{attribute 'linkalways'} 
{attribute 'no_explicit_call' := 'This FB is a CLASS and must be accessed using methods or properties'}
{attribute 'enable_dynamic_creation'}
FUNCTION_BLOCK _WORD EXTENDS DatatypeBase
VAR
	localData : WORD;
	activeData : REFERENCE TO WORD REF= localData;
END_VAR

PROPERTY PUBLIC Address : PVOID
GET
Address := ADR(activeData);
END_GET
END_PROPERTY

METHOD PUBLIC ClearReference
VAR_INPUT
END_VAR
activeData REF= localData;
END_METHOD

METHOD PUBLIC Clone : I_Datatype
VAR
    pClone : POINTER TO _WORD;
END_VAR
pClone := __NEW(_WORD(InitialValue := Value));
Clone := pClone^;
END_METHOD

METHOD FB_init : BOOL
VAR_INPUT
	bInitRetains : BOOL; // if TRUE, the retain variables are initialized (warm start / cold start)
	bInCopyCode : BOOL;  // if TRUE, the instance afterwards gets moved WORDo the copy code (online change)
	InitialValue : WORD;
END_VAR
localData := InitialValue;
END_METHOD

PROPERTY PUBLIC IecType : T_MAXSTRING
GET
IecType := 'WORD';
END_GET
END_PROPERTY

METHOD PUBLIC MakeReferenceTo
VAR_INPUT
	ReferenceTarget : REFERENCE TO WORD;
END_VAR
activeData REF= ReferenceTarget;
END_METHOD

METHOD PUBLIC SerializeWith
VAR_INPUT
	Serializer : I_Serializer;
END_VAR
Serializer.AddWord(activeData);
END_METHOD

PROPERTY PUBLIC Size : UDINT
GET
Size := SIZEOF(activeData);
END_GET
END_PROPERTY

METHOD TryDeserializeFrom : BOOL
VAR_INPUT
	Deserializer : I_Deserializer;
	Feedback : I_DeserializerFeedback;
END_VAR
TryDeserializeFrom := Deserializer.TryGetWord(activeData, Feedback);
END_METHOD

METHOD TryMakeReferenceTo : BOOL
VAR_INPUT
	Target : I_Datatype;
END_VAR
VAR
	pTargetData : POINTER TO WORD;
END_VAR
IF NOT (Target.IecType = IecType) THEN
	RETURN;
END_IF

pTargetData := Target.Address;
activeData REF= pTargetData^;
TryMakeReferenceTo := TRUE;
END_METHOD

PROPERTY PUBLIC Value : WORD
GET
Value := activeData;
END_GET
SET
activeData := Value;
END_SET
END_PROPERTY

END_FUNCTION_BLOCK

(* stored: Version 1.1.0.1, ProductVersion 3.1.4024.12
   POU _WORD: Id {e7bccc65-ec8e-095b-18a1-42a50d575606}, SpecialFunc None
   Folder Constructor: Id {9855b4c7-dd4b-091f-048e-197bbbc3d1ff}
   Property Address: Id {8506bb2c-de33-0776-279b-8f3e62d4e41f}
   Get Get: Id {624c1396-e620-080b-0ec9-5d90a0cf661b}
   Method ClearReference: Id {107fc361-cc8f-01f3-0be2-6be785ad8651}
   Method Clone: Id {24c77b7d-908b-0d82-37f7-3e8e4bfd466a}
   Method FB_init: Id {88882bf8-9a7d-01b3-21ce-f4d80e61d67d}
   Property IecType: Id {aa0f3556-0005-0473-258e-203dbe03d661}
   Get Get: Id {5a893654-cf12-012c-03b2-d2c7473b6d47}
   Method MakeReferenceTo: Id {c68ef1de-2ec4-03cf-262f-3ed89ab93621}
   Method SerializeWith: Id {f1af31b2-031b-0cef-0af3-bc734e479124}
   Property Size: Id {4f1f6c93-bfc9-0181-03ad-e942dcc5d704}
   Get Get: Id {2306413c-09e9-0d25-12a8-21d69e8cb935}
   Method TryDeserializeFrom: Id {c337f86f-3d51-0565-1456-61c27ff55c65}
   Method TryMakeReferenceTo: Id {6584c998-95ea-019d-215d-408811ee36f4}
   Property Value: Id {058c9661-e32a-0fab-0644-75834aa01d79}
   Get Get: Id {0f16fb52-a5db-061a-278c-bb5743ba8ee2}
   Set Set: Id {3a8f4c76-f9ec-099c-21f1-cf58433b5ed9} *)
